       CALL #"Mes_P25_ID2509"
       (
         CM_No := 766 ,
         Tab := 25 ,
         SubTab := 2 ,
         CfgType := 0 ,
         CfgInvert := True ,
         InputRaw := Mes_P25_ID2509_MSG_seq ,
         SC_Local := SL_25_P ,
         CM_ALM := #ALM[757] ,
       );

END_FUNCTION_BLOCK
